// TwinCAT 3 PLC project FSM
// ProgramVersion: 3.1.4026.20
// libraries:
//   Tc2_EtherCAT, * (Beckhoff Automation GmbH)
//   Tc2_Standard, * (Beckhoff Automation GmbH)
//   Tc2_System, * (Beckhoff Automation GmbH)
//   TcUnit, * (www.tcunit.org)
// project tree:
//   DUTs/ E_Command.TcDUT (not stored), E_PodState.TcDUT
//   GVLs/ GVL_FSM.TcGVL, GVL_Levi.TcGVL (not stored), GVL_Prop.TcGVL, GVL_PT.TcGVL (not stored)
//   / PlcTask.TcTTO
//   POUs/FSM/ BasicChecks.TcPOU, CheckCritical.TcPOU (not stored), FB_Charge.TcPOU, FB_Discharge.TcPOU (not stored), FB_Handle_Emergency.TcPOU (not stored), Handle_Movement.TcPOU (not stored), FB_Main_FSM.TcPOU
//   POUs/ MAIN.TcPOU
//   POUs/Tests/ FB_Test_MainFSM.TcPOU
// real-time tasks:
//   TASK PlcTask: cycle T#10ms, priority 20, ADS port 350
//   TASK HeartBeat: cycle T#10ms, priority 1, ADS port 351

CONFIGURATION FSM
    RESOURCE PLC ON TwinCAT3
        TASK PlcTask(INTERVAL := T#10ms, PRIORITY := 20);
        PROGRAM MAIN WITH PlcTask : MAIN;
    END_RESOURCE
END_CONFIGURATION

// ---- DUTs/E_PodState.TcDUT
{attribute 'qualified_only'}
{attribute 'strict'}
{attribute 'to_string'}
TYPE E_PodState :
(
	STATE_EMERGENCY		:= 0,
	STATE_BOOT 			:= 1,
    STATE_SYNC 			:= 2,
    STATE_IDLE 			:= 3,
    STATE_HV_ACTIVE		:= 4,
    STATE_DEMO			:= 5,
    STATE_LEVITATION	:= 6,
    STATE_MOVEMENT		:= 7,
    STATE_MAINTENANCE	:= 8
);
END_TYPE

// ---- GVLs/GVL_FSM.TcGVL
{attribute 'qualified_only'}
VAR_GLOBAL
	enable_heartbeat:		BOOL;
	heartbeat_OK: 			BOOL;
	precharge:				BOOL;
	engage_brakes:			BOOL;
	brakes_engaged:			BOOL;
	enable_levi_checks: 	BOOL;
	enable_prop_checks: 	BOOL;
	enable_temp_checks: 	BOOL;
	safety_inputs_valid: 	BOOL;
	can_bus_ok: 			BOOL;
	ethercat_ready: 		BOOL;
	sdc_closed: 			BOOL;
	critical_temp: 			INT;
	open_SDC: 				BOOL	:= TRUE;
	enable_telemetry: BOOL;
	enable_PT_checks: BOOL;
END_VAR

// ---- GVLs/GVL_Prop.TcGVL
{attribute 'qualified_only'}
VAR_GLOBAL
	speed:					INT;
	target_speed:			INT;
	accelerating:			BOOL;
	braking:				BOOL;
	propulsion_fault: 		BOOL;
	propulsion_enable: 		BOOL;
	propulsion_active: 		BOOL;
	drive_voltages: INT;
END_VAR

// ---- POUs/MAIN.TcPOU
PROGRAM MAIN
VAR
	main_fsm	: FB_Main_FSM;
	main_tests	: FB_Test_MainFSM;
	
	tests_on	: BOOL	:= TRUE;
END_VAR

IF tests_on THEN
	TcUnit.RUN();
ELSE
	main_fsm();
END_IF

END_PROGRAM

// ---- POUs/FSM/FB_Main_FSM.TcPOU
FUNCTION_BLOCK FB_Main_FSM

VAR_INPUT
	currentCmd:					E_Command 	:= E_Command.CMD_NONE;
END_VAR


VAR_OUTPUT
	currentState: 				E_PodState  := E_PodState.STATE_BOOT;
END_VAR

VAR
	criticalFault:				BOOL;
	charging_in_progress:		BOOL;
	discharging_in_progress:	BOOL;
	
	fb_handle_emergency:		FB_Handle_Emergency;
	fb_discharge:				FB_Discharge;
	fb_charge:					FB_Charge;
END_VAR

IF currentCmd = E_Command.CMD_EMERGENCY OR (CheckCritical() AND currentState >= 4) THEN
	currentState := E_PodState.STATE_EMERGENCY;
	criticalFault := TRUE;
	FB_Handle_Emergency();
ELSIF currentState = E_PodState.STATE_MOVEMENT AND 
    GVL_Prop.speed = 0 AND GVL_Prop.target_speed = 0 THEN
		currentState := E_PodState.STATE_LEVITATION;
ELSIF currentState = E_PodState.STATE_DEMO AND GVL_FSM.brakes_engaged THEN
    currentState := E_PodState.STATE_EMERGENCY;
ELSIF currentState = E_PodState.STATE_BOOT AND BasicChecks() THEN
	currentState := E_PodState.STATE_SYNC;
END_IF

CASE currentState OF
	E_PodState.STATE_EMERGENCY:
		IF criticalFault THEN
			FB_Handle_Emergency();
		ELSIF currentCmd = E_Command.CMD_TO_MAINTENANCE THEN
			GVL_FSM.engage_brakes := FALSE;
			currentState := E_PodState.STATE_MAINTENANCE;
		END_IF
		
	E_PodState.STATE_BOOT:  
		IF BasicChecks() THEN
			currentState := E_PodState.STATE_SYNC;
		END_IF
		
	E_PodState.STATE_SYNC:
		GVL_FSM.enable_heartbeat := TRUE;
		IF GVL_FSM.heartbeat_OK AND currentCmd = E_Command.CMD_TO_IDLE THEN
			currentState := E_PodState.STATE_IDLE;
		END_IF
		
	E_PodState.STATE_IDLE:
		// maybe basic checks again WC state - 8
		GVL_FSM.enable_PT_checks := TRUE;
		GVL_FSM.enable_temp_checks := TRUE;
		GVL_FSM.enable_telemetry := TRUE;
		
		IF currentCmd = E_Command.CMD_TO_HV_ACTIVE THEN
			FB_Charge();
			IF GVL_PT.HVAL_STATUS = 1 AND GVL_PT.total_voltage >= 550 THEN
				currentState := E_PodState.STATE_HV_ACTIVE;
			END_IF
		ELSIF currentCmd = E_Command.CMD_TO_MAINTENANCE THEN
			GVL_FSM.engage_brakes := FALSE;
			currentState := E_PodState.STATE_MAINTENANCE;
		END_IF
		
	E_PodState.STATE_HV_ACTIVE:
		GVL_FSM.enable_levi_checks := TRUE;
		GVL_FSM.enable_prop_checks := TRUE;
				
		IF currentCmd = E_Command.CMD_TO_DEMO AND NOT CheckCritical() THEN
			GVL_FSM.engage_brakes := FALSE;
			currentState := E_PodState.STATE_DEMO;
		ELSIF currentCmd = E_Command.CMD_TO_IDLE THEN
			GVL_FSM.open_SDC := TRUE;
			FB_Discharge();
			IF GVL_PT.HVAL_STATUS = 0 AND GVL_Levi.drive_voltages = 0 AND GVL_Prop.drive_voltages = 0 THEN
				currentState := E_PodState.STATE_IDLE;
			END_IF
		END_IF
		
	E_PodState.STATE_DEMO:
		IF currentCmd = E_Command.CMD_TO_IDLE THEN
			GVL_FSM.engage_brakes := TRUE;
			GVL_FSM.open_SDC := TRUE;
			FB_Discharge();
			IF GVL_FSM.brakes_engaged AND GVL_PT.HVAL_STATUS = 0 THEN
				currentState := E_PodState.STATE_IDLE;
			END_IF
		ELSIF currentCmd = E_Command.CMD_TO_LEVITATION THEN
			GVL_Levi.levitation_active := TRUE;
			currentState := E_PodState.STATE_LEVITATION;
		END_IF
		
	E_PodState.STATE_LEVITATION:
		IF currentCmd = E_Command.CMD_TO_DEMO THEN
			GVL_Levi.levitation_active := FALSE;
			currentState := E_PodState.STATE_DEMO;
		ELSIF currentCmd = E_Command.CMD_TO_MOVEMENT THEN
			currentState := E_PodState.STATE_MOVEMENT;
			Handle_movement();
		END_IF
		
	E_PodState.STATE_MOVEMENT:
		Handle_movement();
		
	E_PodState.STATE_MAINTENANCE:
		IF currentCmd = E_Command.CMD_TO_IDLE THEN
			GVL_FSM.engage_brakes := TRUE;
			IF GVL_FSM.brakes_engaged THEN
				currentState := E_PodState.STATE_IDLE;
			END_IF
		END_IF
		
END_CASE

END_FUNCTION_BLOCK

// ---- POUs/FSM/FB_Charge.TcPOU
FUNCTION_BLOCK FB_Charge
VAR_INPUT
END_VAR
VAR_OUTPUT
END_VAR
VAR
END_VAR

END_FUNCTION_BLOCK

// ---- POUs/FSM/BasicChecks.TcPOU
FUNCTION BasicChecks : BOOL
VAR_INPUT
END_VAR
VAR
END_VAR

BasicChecks := 
    GVL_FSM.ethercat_ready AND
    GVL_FSM.safety_inputs_valid AND
    GVL_FSM.can_bus_ok;

END_FUNCTION

// ---- POUs/Tests/FB_Test_MainFSM.TcPOU
FUNCTION_BLOCK FB_Test_MainFSM EXTENDS TcUnit.FB_TestSuite
VAR_INPUT
END_VAR
VAR_OUTPUT
END_VAR
VAR
END_VAR

END_FUNCTION_BLOCK
